% RSLogix 500 project lab 2 Q4 ROBO.RSS, saved by version 8.40.00.08 %
PROJECT "UNTITLED"    % processor: type code 162 %

PROGRAM FILES
  LAD 2   9 rungs

DATA FILES
  S2 STATUS  83 elements
  B3 BINARY  1 elements
  T4 TIMER  1 elements
  C5 COUNTER  1 elements
  R6 CONTROL  1 elements
  N7 INTEGER  1 elements
  F8 FLOAT  1 elements

LADDER 2
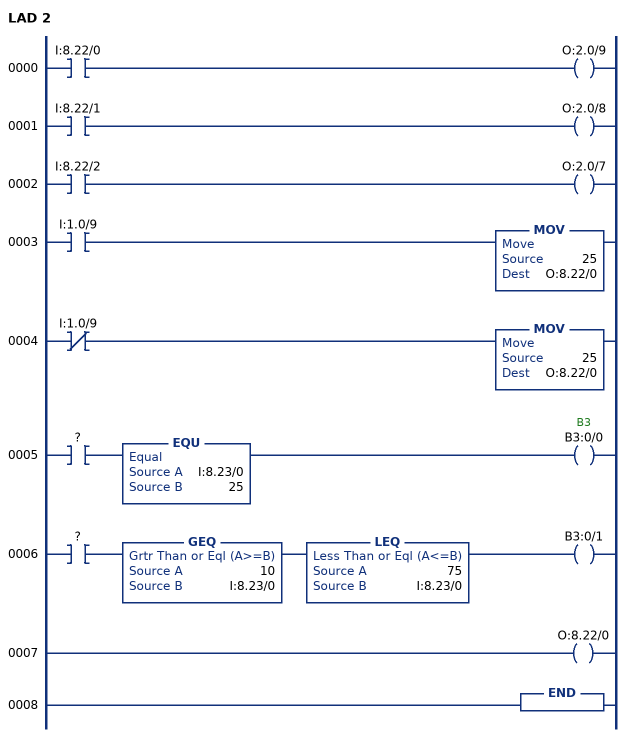
% Rung: 0 %  % edit flag set %
SOR XIC I:8.22/0 OTE O:2.0/9 EOR
% Rung: 1 %  % edit flag set %
SOR XIC I:8.22/1 OTE O:2.0/8 EOR
% Rung: 2 %  % edit flag set %
SOR XIC I:8.22/2 OTE O:2.0/7 EOR
% Rung: 3 %  % edit flag set %
SOR XIC I:1.0/9 MOV 25 O:8.22/0 EOR
% Rung: 4 %  % edit flag set %
SOR XIO I:1.0/9 MOV 25 O:8.22/0 EOR
% Rung: 5 %  % edit flag set %
SOR XIC ? EQU I:8.23/0 25 OTE B3:0/0 EOR
%   B3:0/0  B3 %
% Rung: 6 %  % edit flag set %
SOR XIC ? GEQ 10 I:8.23/0 LEQ 75 I:8.23/0 OTE B3:0/1 EOR
% Rung: 7 %  % edit flag set %
SOR OTE O:8.22/0 EOR
% Rung: 8 %
SOR END EOR
